(*
SPDX-FileCopyrightText: © 2026 Oleksandr Tiutyk <trofimich@gmail.com>
SPDX-License-Identifier: MIT
License: https://opensource.org/license/mit
*)

(*!
<summary>
Beckhoff EL6xxx: 22-byte serial communication input process image.
</summary>
<description>
Encapsulates a 16-bit status word and a 22-byte received data buffer for EL6xxx serial interface terminals.
When used for I/O, link located fields or their containing buffers to the matching selected PDOs.
The record is not a packed wire buffer; compiler padding is not part of the device specification.
Unlinked/default values do not prove valid I/O. The caller evaluates bus/channel validity before use.
Use one owner task per instance and externally synchronize other access; multi-field snapshots are not atomic.
Copies store data without creating hardware links. Keep borrowed field references valid while consumers are bound.
This passive record performs no validation, synchronization, configuration or protocol advancement.
Select the 22-byte serial payload with 16-bit status/control words; larger buffers and 9-bit modes
are outside this model. The owning service implements the transmit/receive toggle handshake.
</description>
*)
TYPE EL6xxx22ByteInData :
STRUCT
	Status : WORD;     
	Data : ARRAY [0..21] OF BYTE; 
END_STRUCT
END_TYPE

(* stored: Version 1.1.0.1, ProductVersion 3.1.4026.18
   DUT EL6xxx22ByteInData: Id {05540d99-a3da-490b-b904-cd3d6478c4c0} *)
